# EPICS autosave request: stdApp/Db/hrSeq_settings.req
# FILE... hrSeq_settings.req
# USAGE.. hrSeq.db fields autosave'd.
$(P)HR$(N)_A1AO.VAL
$(P)HR$(N)_H1AO.VAL
$(P)HR$(N)_K1AO.VAL
$(P)HR$(N)_L1AO.VAL
$(P)HR$(N)_A2AO.VAL
$(P)HR$(N)_H2AO.VAL
$(P)HR$(N)_K2AO.VAL
$(P)HR$(N)_L2AO.VAL
$(P)HR$(N)_EAO.VAL
$(P)HR$(N)_Mode2MO.VAL
$(P)HR$(N)_phi1OffAO.VAL
$(P)HR$(N)_phi2OffAO.VAL
$(P)HR$(N)_ETweakAI.VAL
$(P)HR$(N)_LambdaTweakAI.VAL
$(P)HR$(N)_Theta1TweakAI.VAL
$(P)HR$(N)_Theta2TweakAI.VAL
$(P)HR$(N)_worldTweakAI.VAL
